FUNCTION AngleCutFun : lreal
VAR_INPUT
	angRow:LREAL;
	upper:LREAL;
	lower:LREAL;
	rangLength:LREAL;
END_VAR
VAR
	angCutted:LREAL;
END_VAR

angCutted:=angRow;
WHILE(angCutted>upper OR angCutted<lower) DO
    IF angCutted>upper THEN
        angCutted:=angCutted-rangLength;
    else
        angCutted:=angCutted+rangLength;
    END_IF
END_WHILE
AngleCutFun:=angCutted;

END_FUNCTION

(* stored: Version 1.1.0.1, ProductVersion 3.1.4024.2
   POU AngleCutFun: Id {20341012-9832-4374-a3f9-5c952cab3428}, SpecialFunc None *)
